GLOBALCONSTANTS logiBUS_DO (* Global constants *)
  (* Standard: 61499-1; Description: Copyright (c) 2024 HR Agrartechnik GmbH This program and the accompanying materials are made available under the terms of the Eclipse Public License 2.0 which is available at https://www.eclipse.org/legal/epl-2.0/ SPDX-License-Identifier: EPL-2.0 *)
  (* Version 1.0, 2024-01-25, Franz Höpfinger, HR Agrartechnik GmbH *)
  VAR_GLOBAL CONSTANT
    Output_Q1 : logiBUS_DO_S := (Output := 1);
    Output_Q2 : logiBUS_DO_S := (Output := 2);
    Output_Q3 : logiBUS_DO_S := (Output := 3);
    Output_Q4 : logiBUS_DO_S := (Output := 4);
    Output_Q5 : logiBUS_DO_S := (Output := 5);
    Output_Q6 : logiBUS_DO_S := (Output := 6);
    Output_Q7 : logiBUS_DO_S := (Output := 7);
    Output_Q8 : logiBUS_DO_S := (Output := 8);
    Output_Q9 : logiBUS_DO_S := (Output := 9);
    Invalid : logiBUS_DO_S := (Output := 255);
  END_VAR
END_GLOBALCONSTANTS
